Staubli VAL3: calcTool7En.dtx

num nXPosButTxt[9]
  [2] = 5
  [3] = 10
  [4] = 15
  [5] = 20
  [6] = 25
  [7] = 30
  [8] = 35
num nYPosButTxt = 13
string sUsrMess[120]
  [0] = "Please select a language:"
  [1] = "Creation Tool complex"
  [2] = "This exercise requires:"
  [3] = "- A pointer attached"
  [4] = " to the robot's flange "
  [5] = "- A pointer placed as reference"
  [6] = " inside robot's working envelope "
  [7] = "- Your complex tool"
  [8] = "Press any key to continue..."
  [9] = "Creation of the reference tool"
  [10] = "Length of pointer (mm) :"
  [11] = "Mount the pointer on the robot's flange"
  [12] = "Go to the pointer placed as reference"
  [13] = "Press Enter"
  [14] = "when finish moving the robot"
  [15] = "Creation of your complex tool"
  [16] = "Mount your complex tool"
  [17] = "Go to the reference point "
  [18] = "Values of your tool :"
  [19] = "X :"
  [20] = "Y :"
  [21] = "Z :"
  [22] = "RX :"
  [23] = "RY :"
  [24] = "RZ :"
  [25] = "Verification of calculated TOOL"
  [26] = "Change to Tool mode"
  [27] = "  Select your tool "
  [28] = "Jog the robot in RX RY RZ"
  [29] = "in top of the reference pointer"
  [30] = "Press ESC if the result is not good"
  [31] = "Otherwise press ENTER"
  [32] = "Teaching finished !!!"
  [33] = "-END-"
  [41] = "Creation outil complexe"
  [42] = "Cette manipulation necessite :"
  [43] = "- Une pointe a fixer"
  [44] = " sur la bride du robot"
  [45] = "- Une contre-pointe a fixer"
  [46] = " dans l'enveloppe de travail du robot"
  [47] = "- Votre outil complexe"
  [48] = "Appui sur une touche pour continuer"
  [49] = "Creation de la pointe reference"
  [50] = "Longueur de la Pointe (mm) :"
  [51] = "Monter la pointe sur la bride du robot"
  [52] = "Allez sur la contre-pointe de reference"
  [53] = "Presser Enter"
  [54] = "quand la manipulation est terminee"
  [55] = "Creation de votre outil complexe"
  [56] = "Monter votre outil complexe"
  [57] = "Allez sur la pointe de reference"
  [58] = "Les cotes de votre outil :"
  [59] = "X : "
  [60] = "Y : "
  [61] = "Z : "
  [62] = "RX : "
  [63] = "RY : "
  [64] = "RZ : "
  [65] = "Verification du TOOL calcule"
  [66] = "Passer en mode TOOL"
  [67] = "Selectioner votre outil"
  [68] = "Faire des rotations RX RY RZ"
  [69] = "sur la contre-pointe"
  [70] = "Touche ESC si le resultat n'est pas bon"
  [71] = "Sinon touche ENTER"
  [72] = "L'apprentissage est terminΘ !!!"
  [73] = "-FIN-"
  [81] = "Calculo de herramienta compleja"
  [82] = "Este calculo requiere:"
  [83] = "- Una punta para fijar"
  [84] = "á en la brida del robot."
  [85] = "- Un contra-punta para fijar"
  [86] = "  sobre el area de trabajo del robot."
  [87] = "- La herramienta compleja."
  [88] = "Pulse cualquier tecla para continuar ..."
  [89] = "Creaci≤n herramienta de referencia"
  [90] = "Longitud de la punta (mm):"
  [91] = "Monte la punta en la brida del robot."
  [92] = "Ir a la contra-punta de referencia."
  [93] = "Pulse Intro"
  [94] = "  cuando la manipulaci≤n se acabe."
  [95] = "Creaci≤n de su herramienta compleja "
  [96] = "Ponga su herramienta compleja "
  [97] = "Ir hasta el punto de referencia."
  [98] = "Sφmbolos de la herramienta:"
  [99] = "X:"
  [100] = "Y:"
  [101] = "Z:"
  [102] = "RX:"
  [103] = "RY:"
  [104] = "RZ:"
  [105] = "Verificaci≤n Herramienta calculada"
  [106] = "Poner el robot en modo tool."
  [107] = "Seleccione su  herramienta."
  [108] = "Hacer rotaciones RX RY RZ"
  [109] = "  en la contra-punta"
  [110] = "ESC si el resultado no es correpto."
  [111] = "ENTER  si el resultado es correpto."
  [112] = "El calculo ha terminado!"
  [113] = "-FIN-"
tool tTool = {fatherId=flange[0], ioLink=valve1}
